TYPE "udt_WeldReg_Item"
VERSION : 0.1
// Block: udt_WeldReg_Item
   STRUCT
      Valid : Bool;
      PosBegin : LReal;
      PosEnd : LReal;
      MW_PosBegin : LReal;
      MW_PosEnd : LReal;
   END_STRUCT;

END_TYPE
